FUNCTION_BLOCK TFCiclo_Deposito_Lastra
VAR_INPUT
	Ciclo 		: POINTER TO Stato_Ciclo_Lavoro;
	Programma 	: POINTER TO TFProgramma_Ciclo_Lastra;
	ModuleAX_X 	: POINTER TO TFModulePalletizer_Ax;
	ModuleAX_Y 	: POINTER TO TFModulePalletizer_Ax;
	ModuleAX_Z 	: POINTER TO TFModulePalletizer_Ax;
	ModuleAX_J 	: POINTER TO TFModulePalletizer_AxJ_Lastre;
	ModulePinza : POINTER TO TFModulePalletizer_Pinza;
	StartInterpolazioneAssi : POINTER TO BOOL;
	QuotaPassModePuntoIntermedio : ARRAY [1..3] OF REAL;
	AbilitazioneGlobalePassMode	: BOOL;
	InterrompiCiclo : BOOL;
	Abilita_Ciclo_Step : BOOL;
	Command_Step : BOOL;
	AbilitazioneAnticipoDinamicoMovimenti : BOOL;

END_VAR
VAR_OUTPUT
	STEPDone	: BOOL;
	Errore : UINT;
END_VAR
VAR
	ConAccostamentoZ : BOOL := FALSE;
	StepInto: BOOL;
	PinzaInPresa : BOOL;
	PinzaVerticale : BOOL;
END_VAR

(* Set della variabile che mi permette di fare lo STEP nel ciclo *)
TFTimerCall(ADR(ReMovEjeXCicloDeposito),TimeBase);
StepInto := (Abilita_Ciclo_Step AND Command_Step) OR NOT Abilita_Ciclo_Step;

(* Reset Anticipo Dinamico se non ho l'abilitazione *)
IF NOT AbilitazioneAnticipoDinamicoMovimenti OR NOT HMI_DisabilitaAnticipiGLOBALE THEN
	QuotaAnticipoDinamicaX_Raggiunta := FALSE;
	QuotaAnticipoDinamicaY_Raggiunta := FALSE;
	QuotaAnticipoDinamicaZ_Raggiunta := FALSE;
END_IF

PinzaInPresa 	:= ModulePinza^.StatoPinza.ElementoPrelevato AND  
					ModulePinza^.StatoPinza.LatoDxPiastrellaInPresa AND
					ModulePinza^.StatoPinza.LatoSxPiastrellaInPresa;

PinzaVerticale := NOT(ModuleAX_J^.Ax^.Status.ActPosition > 85 AND ModuleAX_J^.Ax^.Status.ActPosition < 95);

EjeYPosFueraIngombroCargado := TFAsseInFinestra(Posizione_Attuale :=  ModuleAX_Y^.Ax^.Status.ActPosition ,
 Posizione_Finale := Programma_Y[Y_PosFuoriIngombroVuotoLastra].Quota_Destinazione ,FinestraDiControllo := 30.0 );

EjeYPos0Ingombro :=  TFAsseInFinestra(Posizione_Attuale := ModuleAX_Y^.Ax^.Status.ActPosition ,
 Posizione_Finale := Programma_Y[Y_PosPasillo0grados].Quota_Destinazione ,FinestraDiControllo := 30.0 ) ;
 
EjeYPos180Ingombro := TFAsseInFinestra(Posizione_Attuale := ModuleAX_Y^.Ax^.Status.ActPosition ,
 Posizione_Finale := Programma_Y[Y_PosPasillo180grados].Quota_Destinazione ,FinestraDiControllo := 30.0 ) ;
 
 EjeyPosLentaCoger := TFAsseInFinestra(Posizione_Attuale := ModuleAX_Y^.Ax^.Status.ActPosition ,
 Posizione_Finale := Programma_Y[Y_PosStartLentaDepositoLastra].Quota_Destinazione ,FinestraDiControllo := 30.0 ) ;

IF Ciclo^.Passo = 27 THEN

TFTimerSet(ADR(ReMovEjeXCicloDeposito),1000, FALSE );	
ELSE
TFTimerSet(ADR(ReMovEjeX),1000, 
TFAsseInFinestra(Posizione_Attuale := ModuleAX_Y^.Ax^.Status.ActPosition ,
 Posizione_Finale := Programma_Y[Y_PosFuoriIngombroVuotoLastra].Quota_Destinazione ,FinestraDiControllo := 30.0 ) );	
END_IF
  Temp_Bool[69]:=TFAsseInFinestra (Posizione_Attuale := ModuleAX_Y^.Ax^.Status.ActPosition ,
 Posizione_Finale := Programma_Y[Y_PosFuoriIngombroVuotoLastra].Quota_Destinazione ,FinestraDiControllo := 30.0 );
IF NOT InterrompiCiclo THEN
	IF Ciclo^.Stato = TERMINATO OR Ciclo^.Stato = ANNULLATO THEN
		Ciclo^.Passo := 0;
	//ELSIF Ciclo^.Stato = INTERROTTO AND Ciclo^.Passo = 56 THEN
	//	Ciclo^.Passo := 56;
	ELSIF Ciclo^.Stato = INTERROTTO THEN//AND NOT Ciclo^.Passo = 56 THEN
		Ciclo^.Passo := 999;
	END_IF
	Ciclo^.Stato := IN_ESECUZIONE;
	CASE Ciclo^.Passo OF
			(* Case 0 *)
			0:  Ciclo^.Stato := IN_ESECUZIONE;
				Ciclo^.Passo := 10;
				Errore := 0;
				STEPDone := FALSE;
				
			(* Case 10 -  *)
			10:	MaterialeDepositatoSuLinea := FALSE;
				IF PinzaVerticale THEN
					Ciclo^.Passo := 25;
				ELSE
					Ciclo^.Passo := 20;
				END_IF
						
			(* Case 20 - PROGRAMMA[Z_PosFuoriIngombroCaricoLastra] ASSE Z -> TRASLAZIONE A QUOTA DI FUORI INGOMBRO CON lLASTRA A BORDO *)	
			20:	Ciclo^.Stato := IN_ESECUZIONE;
				IF StepInto THEN
					Programma_Z[Z_PosFuoriIngombroCaricoLastra].Stato 			:= DA_ESEGUIRE;
					Programma_Z[Z_PosFuoriIngombroCaricoLastra].InterpolaAsse 	:= NO_INTERPOLAZIONE_ASSE;
					ProgrammaToModule_Z 										:= Programma_Z[Z_PosFuoriIngombroCaricoLastra];
					Ciclo^.Passo := 21;
					STEPDone := FALSE;
				END_IF
				
			(* Case 21 - Attesa completamento del comando MOVETOPOS o del raggiungimento quota di Pre-Movimento se abilitata la funzione*)
			21: 
				IF Programma_Z[Z_PosFuoriIngombroCaricoLastra].Stato = INTERROTTO THEN
					Ciclo^.Passo := 21;		
				ELSIF Programma_Z[Z_PosFuoriIngombroCaricoLastra].Stato = TERMINATO OR
					Asse_Z_InFinestraDiPassMode THEN
					Ciclo^.Passo := 24; //
					STEPDone := TRUE;							
				END_IF
			
			(* Case 22 - Fuori ingombro J - NON usato in questa fase *)	
			22: IF Programma_Z[Z_PosFuoriIngombroCaricoLastra].Stato = INTERROTTO THEN
					 Ciclo^.Passo := 22;
				ELSIF Programma_Z[Z_PosFuoriIngombroCaricoLastra].Stato = TERMINATO OR 
						Asse_Z_InFinestraDiPassMode OR 
						QuotaAnticipoDinamicaZ_Raggiunta THEN
							IF StepInto AND Temp_Bool[3] THEN 
								Programma_J[J_PosFuoriIngombro].Stato 			:= DA_ESEGUIRE;
								Programma_J[J_PosFuoriIngombro].InterpolaAsse 	:= NO_INTERPOLAZIONE_ASSE;
								ProgrammaToModule_J		 						:= Programma_J[J_PosFuoriIngombro];
								Ciclo^.Passo := 23;
								STEPDone := FALSE;
							END_IF									
				END_IF
			
			(* Case 23 - Attesa completamento Fuori ingombro J *)	
			23: IF Programma_Z[Z_PosFuoriIngombroCaricoLastra].Stato = INTERROTTO OR 
					Programma_J[J_PosFuoriIngombro].Stato = INTERROTTO THEN
					 Ciclo^.Passo := 23;
				ELSIF (Programma_Z[Z_PosFuoriIngombroCaricoLastra].Stato = TERMINATO OR Asse_Z_InFinestraDiPassMode (*OR QuotaAnticipoDinamicaZ_Raggiunta*)) AND 
					(Programma_J[J_PosFuoriIngombro].Stato = TERMINATO OR Asse_J_InFinestraDiPassMode OR QuotaAnticipoDinamicaJ_Raggiunta) THEN
						Ciclo^.Passo := 24;
						STEPDone := TRUE;										
				END_IF	
							
				
			(* Case 24 - Scelgo in quale direzione devo muovermi per primo a seconda della disposizione delle postazioni *)	
			24:	
				IF Programma_Z[Z_PosFuoriIngombroCaricoLastra].Stato = INTERROTTO THEN
					Ciclo^.Passo := 21;	
				ELSE
					Ciclo^.Passo := 25;
				END_IF
					
		{Region "Dipsoizione postazioni lungo X"}		
			(* Case 25 - Vado a quota di fuori ingombro con Y e J *)
			25:	
						Temp_Bool[84] := ((WorkAreaState[PosRobot].Supporto.Tipologia = CAVALLETTO AND 
							workAreaState[Mission.PPlace].Supporto.Tipologia = BUNDLE)  OR MultiplesCavalletesReceta ) AND PosicionJOrigen <> PosicionJDestino  ;
					
				IF StepInto THEN
					IF PinzaVerticale THEN
						Programma_Z[Z_PosFuoriIngombroCaricoLastra].Stato 			:= DA_ESEGUIRE;
						Programma_Z[Z_PosFuoriIngombroCaricoLastra].InterpolaAsse 	:= INTERPOLAZIONE_ASSE;
						ProgrammaToModule_Z 										:= Programma_Z[Z_PosFuoriIngombroCaricoLastra];
					END_IF
					
					IF WorkAreaState[PosRobot].Supporto.Tipologia = BUNDLE  AND Programma_J[J_PosFuoriIngombro].Quota_Destinazione = 0 THEN
						(*
						//**********************************************************************
						Programma_Y[Y_PosPasillo0grados].Stato 				:= NON_ESEGUITO;
						Programma_Y[Y_PosPasillo180grados].Stato 			:= NON_ESEGUITO;
						Programma_Y[Y_PosFuoriIngombroCaricoLastra].Stato 	:= NON_ESEGUITO;
						//********************************************************************
						*)
  						Programma_Y[Y_PosgiroPieza].Stato 			:= DA_ESEGUIRE;
						Programma_Y[Y_PosgiroPieza].InterpolaAsse 	:= INTERPOLAZIONE_ASSE;
						ProgrammaToModule_Y 						:= Programma_Y[Y_PosgiroPieza];
						IF Temp_Bool[2] THEN 
							Ciclo^.Passo := 27;
							STEPDone := FALSE;
						END_IF
					ELSIF ((WorkAreaState[PosRobot].Supporto.Tipologia = CAVALLETTO AND 
							workAreaState[Mission.PPlace].Supporto.Tipologia = BUNDLE)  OR MultiplesCavalletesReceta ) AND  NuEstacionPiking <> 0  
								 THEN
							IF PosicionJActual = 0 THEN
								Programma_Y[Y_PosPasillo0grados].Stato 			:= DA_ESEGUIRE;
								Programma_Y[Y_PosPasillo0grados].InterpolaAsse 	:= INTERPOLAZIONE_ASSE;
								ProgrammaToModule_Y 							:= Programma_Y[Y_PosPasillo0grados];
								IF Temp_Bool[10] AND EjeYPos0Ingombro THEN 
									Ciclo^.Passo := 60;
									STEPDone := FALSE;
								END_IF
							END_IF
							IF PosicionJActual = 180  THEN
								Programma_Y[Y_PosPasillo180grados].Stato 			:= DA_ESEGUIRE;
								Programma_Y[Y_PosPasillo180grados].InterpolaAsse 	:= INTERPOLAZIONE_ASSE;
								ProgrammaToModule_Y 								:= Programma_Y[Y_PosPasillo180grados];
								IF Temp_Bool[10]AND EjeYPos180Ingombro THEN 
									Ciclo^.Passo := 60;
									STEPDone := FALSE;
								END_IF
							END_IF
							
							IF PosicionJActual = 90 THEN
								IF PosicionJDestino = 0 THEN
									Programma_Y[Y_PosPasillo0grados].Stato 			:= DA_ESEGUIRE;
									Programma_Y[Y_PosPasillo0grados].InterpolaAsse 	:= INTERPOLAZIONE_ASSE;
									ProgrammaToModule_Y 							:= Programma_Y[Y_PosPasillo0grados];
									
									Programma_J[Pos0TrasporteCavallete].Stato 						:= DA_ESEGUIRE;
									Programma_J[Pos0TrasporteCavallete].InterpolaAsse 				:= INTERPOLAZIONE_ASSE;
									ProgrammaToModule_J		 									:= Programma_J[Pos0TrasporteCavallete];
									
									IF Temp_Bool[10] AND EjeYPos0Ingombro THEN 
										Ciclo^.Passo := 60;
										STEPDone := FALSE;
									END_IF
								END_IF
								
								IF PosicionJDestino = 180  THEN
									Programma_Y[Y_PosPasillo180grados].Stato 			:= DA_ESEGUIRE;
									Programma_Y[Y_PosPasillo180grados].InterpolaAsse 	:= INTERPOLAZIONE_ASSE;
									ProgrammaToModule_Y 								:= Programma_Y[Y_PosPasillo180grados];
									
									Programma_J[Pos180TrasporteCavallete].Stato 						:= DA_ESEGUIRE;
									Programma_J[Pos180TrasporteCavallete].InterpolaAsse 				:= INTERPOLAZIONE_ASSE;
									ProgrammaToModule_J		 									:= Programma_J[Pos180TrasporteCavallete];
									
									IF Temp_Bool[10] AND EjeYPos180Ingombro THEN 
										Ciclo^.Passo := 60;
										STEPDone := FALSE;
									END_IF
								END_IF
								IF PosicionJDestino = 90  THEN//*************************************************
									Programma_Y[Y_PosFuoriIngombroCaricoLastra].Stato 			:= DA_ESEGUIRE;
									Programma_Y[Y_PosFuoriIngombroCaricoLastra].InterpolaAsse 	:= INTERPOLAZIONE_ASSE;
									ProgrammaToModule_Y 										:= Programma_Y[Y_PosFuoriIngombroCaricoLastra];
									
									
									Programma_J[J_PosFuoriIngombro].Stato 						:= DA_ESEGUIRE;
									Programma_J[J_PosFuoriIngombro].InterpolaAsse 				:= INTERPOLAZIONE_ASSE;
									ProgrammaToModule_J		 									:= Programma_J[J_PosFuoriIngombro];
									
									StartInterpolazioneAssi^ := TRUE; //Abilito l'interpolazione degli assi						
									IF Temp_Bool[90] THEN 
											Ciclo^.Passo := 26;
											STEPDone := FALSE;
									END_IF
								END_IF
							END_IF
						
					
						
							
					ELSIF (((WorkAreaState[PosRobot].Supporto.Tipologia = CAVALLETTO AND 
							workAreaState[Mission.PPlace].Supporto.Tipologia = BUNDLE ) OR MultiplesCavalletesReceta) AND PosicionJOrigen = PosicionJDestino ) OR 
								(WorkAreaState[PosRobot].Supporto.Tipologia = CASSA_STANDARD AND 	
								WorkAreaState[Mission.PPlace].Supporto.Tipologia = CASSA_STANDARD AND 
									PosicionJActual = PosicionJDestino ) 
								 												THEN
						(*
						//********************************************************************++
						Programma_Y[Y_PosPasillo0grados].Stato 				:= NON_ESEGUITO;
						Programma_Y[Y_PosPasillo180grados].Stato 			:= NON_ESEGUITO;
						Programma_Y[Y_PosgiroPieza].Stato 					:= NON_ESEGUITO;		 
						//********************************************************************++	
						*)	 
						Programma_Y[Y_PosFuoriIngombroCaricoLastra].Stato 			:= DA_ESEGUIRE;
						Programma_Y[Y_PosFuoriIngombroCaricoLastra].InterpolaAsse 	:= INTERPOLAZIONE_ASSE;
						ProgrammaToModule_Y 										:= Programma_Y[Y_PosFuoriIngombroCaricoLastra];
						
						
						Programma_J[J_PosFuoriIngombro].Stato 						:= DA_ESEGUIRE;
						Programma_J[J_PosFuoriIngombro].InterpolaAsse 				:= INTERPOLAZIONE_ASSE;
						ProgrammaToModule_J		 									:= Programma_J[J_PosFuoriIngombro];
						
						StartInterpolazioneAssi^ := TRUE; //Abilito l'interpolazione degli assi						
						IF Temp_Bool[90] THEN 
						Ciclo^.Passo := 26;
						STEPDone := FALSE;
						END_IF
					ELSIF workAreaState[PosRobot].Supporto.Tipologia = BUNDLE  AND  PosicionJOrigen = PosicionJDestino  
								 THEN
						(*
						//********************************************************************++
						Programma_Y[Y_PosPasillo0grados].Stato 				:= NON_ESEGUITO;
						Programma_Y[Y_PosPasillo180grados].Stato 			:= NON_ESEGUITO;
						Programma_Y[Y_PosgiroPieza].Stato 					:= NON_ESEGUITO;		 
						//********************************************************************++
						*)	
						Programma_Y[Y_PosFuoriIngombroCaricoLastra].Stato 			:= DA_ESEGUIRE;
						Programma_Y[Y_PosFuoriIngombroCaricoLastra].InterpolaAsse 	:= INTERPOLAZIONE_ASSE;
						ProgrammaToModule_Y 										:= Programma_Y[Y_PosFuoriIngombroCaricoLastra];
						
						
						Programma_J[J_PosFuoriIngombro].Stato 						:= DA_ESEGUIRE;
						Programma_J[J_PosFuoriIngombro].InterpolaAsse 				:= INTERPOLAZIONE_ASSE;
						ProgrammaToModule_J		 									:= Programma_J[J_PosFuoriIngombro];
						
						StartInterpolazioneAssi^ := TRUE; //Abilito l'interpolazione degli assi						
						IF Temp_Bool[90] THEN 
						Ciclo^.Passo := 26;
						STEPDone := FALSE;
						END_IF
					ELSE
						(*
						//********************************************************************++
						Programma_Y[Y_PosPasillo0grados].Stato 				:= NON_ESEGUITO;
						Programma_Y[Y_PosPasillo180grados].Stato 			:= NON_ESEGUITO;
						Programma_Y[Y_PosgiroPieza].Stato 					:= NON_ESEGUITO;		 
						//********************************************************************++
						*)	
						Programma_Y[Y_PosFuoriIngombroCaricoLastra].Stato 			:= DA_ESEGUIRE;
						Programma_Y[Y_PosFuoriIngombroCaricoLastra].InterpolaAsse 	:= INTERPOLAZIONE_ASSE;
						ProgrammaToModule_Y 										:= Programma_Y[Y_PosFuoriIngombroCaricoLastra];
						
						
						Programma_J[J_PosFuoriIngombro].Stato 						:= DA_ESEGUIRE;
						Programma_J[J_PosFuoriIngombro].InterpolaAsse 				:= INTERPOLAZIONE_ASSE;
						ProgrammaToModule_J		 									:= Programma_J[J_PosFuoriIngombro];
						
						StartInterpolazioneAssi^ := TRUE; //Abilito l'interpolazione degli assi						
						IF Temp_Bool[90] THEN 
						Ciclo^.Passo := 26;
						STEPDone := FALSE;
						END_IF
					END_IF 
					
				END_IF
					
					
				
			// VOY CON X A LA POSICION DE DEPOSITO
			60: 	IF 
 						(Programma_Y[Y_PosPasillo0grados].Stato 				= INTERROTTO AND PosicionJActual = 0) OR 
						(Programma_Y[Y_PosPasillo180grados].Stato 			= INTERROTTO AND PosicionJActual = 180 )OR 
						Programma_Z[Z_PosFuoriIngombroCaricoLastra].Stato 	= INTERROTTO OR 
						Programma_J[J_PosSfogliatura].Stato 				= INTERROTTO THEN
						Ciclo^.Passo := 60;
					ELSE	
						IF  ((Programma_Y[Y_PosPasillo0grados].Stato 				= TERMINATO AND PosicionJActual = 0) OR  
							(Programma_Y[Y_PosPasillo180grados].Stato 			= TERMINATO AND PosicionJActual = 180)) AND
							Programma_Z[Z_PosFuoriIngombroCaricoLastra].Stato 	= TERMINATO AND
							Programma_J[J_PosSfogliatura].Stato 				= TERMINATO THEN
								 	
							IF 	NOT MultiplesCavalletesReceta OR PosicionJDestino = 90 OR (WorkAreaState[Mission.PPlace].Supporto.Tipologia = BUNDLE AND MultiplesCavalletesReceta) THEN	
							Programma_X[X_PosStartLentaDepositoLastra].Stato 			:= DA_ESEGUIRE;
							Programma_X[X_PosStartLentaDepositoLastra].InterpolaAsse 	:= NO_INTERPOLAZIONE_ASSE;
							ProgrammaToModule_X 										:= Programma_X[X_PosStartLentaDepositoLastra];
							ELSE 
								Programma_X[X_PosGiroPiezaTraCavallete].Stato 			:= DA_ESEGUIRE;
								Programma_X[X_PosGiroPiezaTraCavallete].InterpolaAsse 	:= NO_INTERPOLAZIONE_ASSE;
								ProgrammaToModule_X 										:= Programma_X[X_PosGiroPiezaTraCavallete];
							END_IF
							IF Temp_Bool[11] THEN 
								Ciclo^.Passo := 61;
								STEPDone := FALSE;	
							END_IF
						END_IF 
					END_IF	
			 // VPY CON Y A LA POSICION DE GIRAR		
					
			61: 	IF (Programma_Y[Y_PosFuoriIngombroCaricoLastra].Stato 	= INTERROTTO AND ProgramaEjes.EjeY = 127)  OR 
						(Programma_Y[Y_PosPasillo0grados].Stato 				= INTERROTTO  AND  PosicionJActual = 0 AND ProgramaEjes.EjeY = 128 )OR
						(Programma_Y[Y_PosPasillo180grados].Stato 				= INTERROTTO  AND  PosicionJActual = 180 AND  ProgramaEjes.EjeY = 129)OR
						Programma_Z[Z_PosFuoriIngombroCaricoLastra].Stato 		= INTERROTTO OR 
						Programma_J[J_PosSfogliatura].Stato 					= INTERROTTO OR
						(Programma_X[X_PosStartLentaDepositoLastra].Stato 		= INTERROTTO AND ProgramaEjes.EjeX = 104) OR 
						(Programma_X[X_PosGiroPiezaTraCavallete].Stato 			= INTERROTTO AND  ProgramaEjes.EjeX = 127) 	THEN
						Ciclo^.Passo := 60;
					ELSE	
						IF ((Programma_Y[Y_PosFuoriIngombroCaricoLastra].Stato =  TERMINATO AND ProgramaEjes.EjeY = 127 )OR
							(Programma_Y[Y_PosPasillo0grados].Stato =  TERMINATO AND   PosicionJActual = 0 AND ProgramaEjes.EjeY = 128) OR
							(Programma_Y[Y_PosPasillo180grados].Stato =  TERMINATO AND  PosicionJActual = 180 AND ProgramaEjes.EjeY = 129 ))
							AND	Programma_Z[Z_PosFuoriIngombroCaricoLastra].Stato = TERMINATO 
								AND	Programma_J[J_PosSfogliatura].Stato = TERMINATO
									AND ((Programma_X[X_PosStartLentaDepositoLastra].Stato =TERMINATO AND ProgramaEjes.EjeX = 104) OR
									 (Programma_X[X_PosGiroPiezaTraCavallete].Stato =TERMINATO AND ProgramaEjes.EjeX = 127 )) AND PosicionJDestino <> 90 		THEN
									 
									 
								IF (Programma_X[X_PosGiroPiezaTraCavallete].Stato =TERMINATO AND ProgramaEjes.EjeX = 127) OR  
									(Programma_X[X_PosStartLentaDepositoLastra].Stato 		= TERMINATO AND ProgramaEjes.EjeX = 104 AND PosicionJActual <> PosicionJDestino)		THEN
									Programma_Y[Y_PosgiroPieza].Stato 			:= DA_ESEGUIRE;
									Programma_Y[Y_PosgiroPieza].InterpolaAsse 	:= INTERPOLAZIONE_ASSE;
									ProgrammaToModule_Y 						:= Programma_Y[Y_PosgiroPieza];
									IF Temp_Bool[12] THEN 
										Ciclo^.Passo := 62;
										STEPDone := FALSE;	
									END_IF
									ELSIF Programma_X[X_PosStartLentaDepositoLastra].Stato 		= TERMINATO AND ProgramaEjes.EjeX = 104 and PosicionJActual = PosicionJDestino THEN 
									IF Temp_Bool[12] THEN 
										Ciclo^.Passo := 31;
										STEPDone := FALSE;	
									END_IF	
								END_IF
							ELSIF  ((Programma_Y[Y_PosFuoriIngombroCaricoLastra].Stato =  TERMINATO AND ProgramaEjes.EjeY = 127 )OR
										(Programma_Y[Y_PosPasillo0grados].Stato =  TERMINATO AND   PosicionJActual = 0 AND ProgramaEjes.EjeY = 128) OR
											(Programma_Y[Y_PosPasillo180grados].Stato =  TERMINATO AND  PosicionJActual = 180 AND ProgramaEjes.EjeY = 129 ))
													AND	Programma_Z[Z_PosFuoriIngombroCaricoLastra].Stato = TERMINATO 
															AND	Programma_J[J_PosSfogliatura].Stato = TERMINATO
																AND ((Programma_X[X_PosStartLentaDepositoLastra].Stato =TERMINATO AND ProgramaEjes.EjeX = 104) OR
									 								(Programma_X[X_PosGiroPiezaTraCavallete].Stato =TERMINATO AND ProgramaEjes.EjeX = 127 )) AND PosicionJDestino = 90	 THEN 
										IF Temp_Bool[12] THEN 
										Ciclo^.Passo := 31;
										STEPDone := FALSE;	
									END_IF						
						END_IF 
					END_IF	
			62: 	IF Programma_Y[Y_PosgiroPieza].Stato 	= INTERROTTO  OR 
						Programma_Z[Z_PosFuoriIngombroCaricoLastra].Stato 	= INTERROTTO OR 
						Programma_J[J_PosSfogliatura].Stato 				= INTERROTTO OR
						Programma_X[X_PosStartLentaDepositoLastra].Stato 	= INTERROTTO AND NOT MultiplesCavalletesReceta OR 
						Programma_X[X_PosGiroPiezaTraCavallete].Stato 	= INTERROTTO AND MultiplesCavalletesReceta	 THEN
						Ciclo^.Passo := 62;
					ELSE	
						IF Programma_Y[Y_PosgiroPieza].Stato =  TERMINATO 	
								AND	Programma_Z[Z_PosFuoriIngombroCaricoLastra].Stato = TERMINATO 
									AND	Programma_J[J_PosSfogliatura].Stato = TERMINATO
									AND Programma_X[X_PosStartLentaDepositoLastra].Stato =TERMINATO AND NOT MultiplesCavalletesReceta OR 	
										Programma_X[X_PosGiroPiezaTraCavallete].Stato =TERMINATO AND  MultiplesCavalletesReceta	THEN
							Programma_J[J_PosFuoriIngombro].Stato 						:= DA_ESEGUIRE;
							Programma_J[J_PosFuoriIngombro].InterpolaAsse 				:= INTERPOLAZIONE_ASSE;
							ProgrammaToModule_J		 									:= Programma_J[J_PosFuoriIngombro];
							IF Temp_Bool[13] THEN 
								Ciclo^.Passo := 63;
								STEPDone := FALSE;	
							END_IF
						END_IF 
					END_IF	
			63: 	IF Programma_Y[Y_PosgiroPieza].Stato 	= INTERROTTO  OR 
						Programma_Z[Z_PosFuoriIngombroCaricoLastra].Stato 	= INTERROTTO OR 
						Programma_J[J_PosFuoriIngombro].Stato 				= INTERROTTO OR
						Programma_X[X_PosStartLentaDepositoLastra].Stato 	= INTERROTTO AND NOT MultiplesCavalletesReceta OR
						Programma_X[X_PosGiroPiezaTraCavallete].Stato =INTERROTTO AND  MultiplesCavalletesReceta THEN
						Ciclo^.Passo := 63;
					ELSE	
						IF Programma_Y[Y_PosgiroPieza].Stato =  TERMINATO 	
								AND	Programma_Z[Z_PosFuoriIngombroCaricoLastra].Stato = TERMINATO 
									AND	Programma_J[J_PosFuoriIngombro].Stato = TERMINATO
									AND (Programma_X[X_PosStartLentaDepositoLastra].Stato =TERMINATO AND NOT MultiplesCavalletesReceta) OR
									(Programma_X[X_PosGiroPiezaTraCavallete].Stato = TERMINATO AND  MultiplesCavalletesReceta )	THEN
						(*
						//********************************************************************++
						Programma_Y[Y_PosPasillo0grados].Stato 				:= NON_ESEGUITO;
						Programma_Y[Y_PosPasillo180grados].Stato 			:= NON_ESEGUITO;
						Programma_Y[Y_PosgiroPieza].Stato 					:= NON_ESEGUITO;		 
						//********************************************************************++
						*)	
							Programma_Y[Y_PosFuoriIngombroCaricoLastra].Stato 			:= DA_ESEGUIRE;
							Programma_Y[Y_PosFuoriIngombroCaricoLastra].InterpolaAsse 	:= INTERPOLAZIONE_ASSE;
							ProgrammaToModule_Y 										:= Programma_Y[Y_PosFuoriIngombroCaricoLastra];
							IF Temp_Bool[14] THEN 
								Ciclo^.Passo := 64;
								STEPDone := FALSE;	
							END_IF
						END_IF 
					END_IF	
			64 :
				 IF Programma_X[X_PosStartLentaDepositoLastra].Stato = INTERROTTO AND NOT MultiplesCavalletesReceta OR
					Programma_X[X_PosGiroPiezaTraCavallete].Stato = INTERROTTO AND  MultiplesCavalletesReceta OR 
					Programma_Y[Y_PosFuoriIngombroCaricoLastra].Stato = INTERROTTO OR
					Programma_Z[Z_PosFuoriIngombroCaricoLastra].Stato = INTERROTTO OR 
					Programma_J[J_PosFuoriIngombro].Stato = INTERROTTO THEN
						Ciclo^.Passo := 64;
				ELSE	
						IF (Programma_Y[Y_PosFuoriIngombroCaricoLastra].Stato =  TERMINATO AND ProgramaEjes.EjeY = 126) AND 	
							Programma_Z[Z_PosFuoriIngombroCaricoLastra].Stato = TERMINATO AND
							Programma_J[J_PosFuoriIngombro].Stato = TERMINATO AND 
									((Programma_X[X_PosStartLentaDepositoLastra].Stato =TERMINATO AND NOT MultiplesCavalletesReceta) OR
									(Programma_X[X_PosGiroPiezaTraCavallete].Stato = TERMINATO AND  MultiplesCavalletesReceta ) )AND  Temp_Bool[69] AND  Temp_Bool[70]	THEN
							Programma_X[X_PosStartLentaDepositoLastra].Stato 			:= DA_ESEGUIRE;
							Programma_X[X_PosStartLentaDepositoLastra].InterpolaAsse 	:= NO_INTERPOLAZIONE_ASSE;
							ProgrammaToModule_X 										:= Programma_X[X_PosStartLentaDepositoLastra];
							IF Temp_Bool[18] THEN 
								Ciclo^.Passo := 31;
								STEPDone := FALSE;	
							END_IF
						END_IF 
				END_IF	
			
					
			27: 	IF Programma_Y[Y_PosgiroPieza].Stato 	= INTERROTTO  OR 
						Programma_Z[Z_PosFuoriIngombroCaricoLastra].Stato 	= INTERROTTO OR 
						Programma_J[J_PosFuoriIngombro].Stato 				= INTERROTTO THEN
						Ciclo^.Passo := 27;
					ELSE	
						IF Programma_Y[Y_PosgiroPieza].Stato =  TERMINATO 		THEN
							Programma_J[J_PosFuoriIngombro].Stato 						:= DA_ESEGUIRE;
							Programma_J[J_PosFuoriIngombro].InterpolaAsse 				:= No_INTERPOLAZIONE_ASSE;
							ProgrammaToModule_J		 									:= Programma_J[J_PosFuoriIngombro];
							IF Temp_Bool[11] THEN 
							Ciclo^.Passo := 28;
							STEPDone := FALSE;	
					END_IF
						END_IF 
					END_IF
					
			28: 	IF Programma_Y[Y_PosgiroPieza].Stato 	= INTERROTTO  OR 
						Programma_Z[Z_PosFuoriIngombroCaricoLastra].Stato 	= INTERROTTO OR 
						Programma_J[J_PosFuoriIngombro].Stato 				= INTERROTTO THEN
						Ciclo^.Passo := 27;
					ELSE	
						IF Programma_Y[Y_PosgiroPieza].Stato =  TERMINATO AND Programma_J[J_PosFuoriIngombro].Stato = TERMINATO	 	THEN
							
						(*
						//********************************************************************++
						Programma_Y[Y_PosPasillo0grados].Stato 				:= NON_ESEGUITO;
						Programma_Y[Y_PosPasillo180grados].Stato 			:= NON_ESEGUITO;
						Programma_Y[Y_PosgiroPieza].Stato 					:= NON_ESEGUITO;		 
						//********************************************************************++
						*)	
							Programma_Y[Y_PosFuoriIngombroCaricoLastra].Stato 			:= DA_ESEGUIRE;
							Programma_Y[Y_PosFuoriIngombroCaricoLastra].InterpolaAsse 	:= INTERPOLAZIONE_ASSE;
							ProgrammaToModule_Y 										:= Programma_Y[Y_PosFuoriIngombroCaricoLastra];
							IF Temp_Bool[12] THEN 
							Ciclo^.Passo := 26;
							STEPDone := FALSE;	
							END_IF
						END_IF 
					END_IF
					
			(* Case 26 - Check se a quota di fuori ingombro con Y & J *)		
			26:	IF Programma_Y[Y_PosFuoriIngombroCaricoLastra].Stato 	= INTERROTTO OR 
					Programma_Z[Z_PosFuoriIngombroCaricoLastra].Stato 	= INTERROTTO OR 
					Programma_J[J_PosFuoriIngombro].Stato 				= INTERROTTO THEN
						Ciclo^.Passo := 26;
				ELSE	
				IF WorkAreaState[PosRobot].Supporto.Tipologia = BUNDLE  AND Programma_J[J_PosFuoriIngombro].Quota_Destinazione = 0 THEN
					IF  Programma_Y[Y_PosFuoriIngombroCaricoLastra].Stato = TERMINATO  AND
						Programma_J[J_PosFuoriIngombro].Stato = TERMINATO  AND
						Programma_Z[Z_PosFuoriIngombroCaricoLastra].Stato = TERMINATO THEN
						IF Temp_Bool[91] THEN 
						Ciclo^.Passo := 30;
						STEPDone := TRUE;	
						END_IF						
					END_IF
				ELSE
					IF (Programma_Y[Y_PosFuoriIngombroCaricoLastra].Stato = TERMINATO OR Asse_Y_InFinestraDiPassMode OR QuotaAnticipoDinamicaY_Raggiunta) AND
						(Programma_J[J_PosFuoriIngombro].Stato = TERMINATO OR Asse_J_InFinestraDiPassMode OR QuotaAnticipoDinamicaJ_Raggiunta) AND
						Programma_Z[Z_PosFuoriIngombroCaricoLastra].Stato = TERMINATO THEN
						IF Temp_Bool[92] THEN 
						Ciclo^.Passo := 30;
						STEPDone := TRUE;	
						END_IF
					END_IF
				END_IF	
				END_IF
										
			(* Case 30 - PROGRAMMA[0] ASSE X  -> TRASLAZIONE A QUOTA DI DEPOSITO  *)	
			30:	IF Programma_Z[Z_PosFuoriIngombroCaricoLastra].Stato = INTERROTTO OR 
					Programma_Y[Y_PosFuoriIngombroCaricoLastra].Stato = INTERROTTO OR 
					Programma_J[J_PosFuoriIngombro].Stato = INTERROTTO THEN
						Ciclo^.Passo := 30;										
				ELSE
					IF StepInto THEN
						Programma_X[X_PosStartLentaDepositoLastra].Stato 			:= DA_ESEGUIRE;
						Programma_X[X_PosStartLentaDepositoLastra].InterpolaAsse 	:= NO_INTERPOLAZIONE_ASSE;
						ProgrammaToModule_X 										:= Programma_X[X_PosStartLentaDepositoLastra];
						IF Temp_Bool[93] THEN 
						Ciclo^.Passo := 31;
						STEPDone := FALSE;
						END_IF
					END_IF
				END_IF			
			
			(* Case 31 -  Attesa completamento del comando MOVETOPOS o del raggiungimento quota di Pre-Movimento se abilitata la funzione *)
			31: 
				IF Programma_X[X_PosStartLentaDepositoLastra].Stato = INTERROTTO   OR
					(Programma_Y[Y_PosFuoriIngombroCaricoLastra].Stato = INTERROTTO AND  ProgramaEjes.EjeY = 126 ) OR
					(Programma_Y[Y_PosPasillo0grados].Stato = INTERROTTO AND  ProgramaEjes.EjeY = 128)  OR
					(Programma_Y[Y_PosPasillo180grados].Stato = INTERROTTO AND  ProgramaEjes.EjeY = 129)  OR
					Programma_Z[Z_PosFuoriIngombroCaricoLastra].Stato = INTERROTTO OR 
					Programma_J[J_PosFuoriIngombro].Stato = INTERROTTO THEN
						Ciclo^.Passo := 31;
				ELSE	
					IF (Programma_X[X_PosStartLentaDepositoLastra].Stato = TERMINATO OR Asse_X_InFinestraDiPassMode OR QuotaAnticipoDinamicaX_Raggiunta) THEN 
						IF WorkAreaState[Mission.PPlace].Supporto.Tipologia <> CAVALLETTO AND WorkAreaState[Mission.PPlace].Supporto.Tipologia <> BUNDLE THEN //se non devo depositare nel cavalletto...	
							Ciclo^.Passo := 32;//ciclo per orizzontale
						ELSE
							Ciclo^.Passo := 40;//Ciclo per cavalletto
						END_IF
						STEPDone := TRUE;							
					END_IF
				END_IF
				
			(* Case 32 - Vado a quota di START LENTA CON GLI ASSI con Y,Z,J *)
			32:
				IF Programma_X[X_PosStartLentaDepositoLastra].Stato = INTERROTTO OR
					(Programma_Y[Y_PosFuoriIngombroCaricoLastra].Stato = INTERROTTO AND  ProgramaEjes.EjeY = 126 ) OR
					(Programma_Y[Y_PosPasillo0grados].Stato = INTERROTTO AND  ProgramaEjes.EjeY = 128)  OR
					(Programma_Y[Y_PosPasillo180grados].Stato = INTERROTTO AND  ProgramaEjes.EjeY = 129)  OR
					Programma_Z[Z_PosFuoriIngombroCaricoLastra].Stato = INTERROTTO OR 
					Programma_J[J_PosFuoriIngombro].Stato = INTERROTTO THEN
						Ciclo^.Passo := 32;										
				ELSE
					IF StepInto AND Programma_X[X_PosStartLentaDepositoLastra].Stato = TERMINATO  THEN
						TFParametersArrayClear(ADR(ParametersArray));
						Programma_Y[Y_PosStartLentaDepositoLastra].Stato 			:= DA_ESEGUIRE;
						Programma_Y[Y_PosStartLentaDepositoLastra].InterpolaAsse 	:= INTERPOLAZIONE_ASSE;
						ProgrammaToModule_Y 										:= Programma_Y[Y_PosStartLentaDepositoLastra];
				
						//Programma_Z[Z_PosStartLentaDepositoLastra].Stato 			:= DA_ESEGUIRE;
						//Programma_Z[Z_PosStartLentaDepositoLastra].InterpolaAsse 	:= INTERPOLAZIONE_ASSE;
						//ProgrammaToModule_Z 										:= Programma_Z[Z_PosStartLentaDepositoLastra];
						
						Programma_J[J_PosDepositoLastra].Stato 						:= DA_ESEGUIRE;
						Programma_J[J_PosDepositoLastra].InterpolaAsse 				:= INTERPOLAZIONE_ASSE;
						ProgrammaToModule_J 										:= Programma_J[J_PosDepositoLastra];
						
						StartInterpolazioneAssi^ := TRUE; //Abilito l'interpolazione degli assi
												
						Ciclo^.Passo := 33;
						STEPDone := FALSE;
					END_IF
				END_IF
			
			(* Case 33 - Attendo completamento comando o assi in finsetra *)
			33:
				IF Programma_Y[Y_PosStartLentaDepositoLastra].Stato 	= TERMINATO OR ((Asse_Y_InFinestraDiPassMode OR TRUE) AND WorkAreaState[Mission.PPlace].Supporto.Tipologia <> CAVALLETTO AND WorkAreaState[Mission.PPlace].Supporto.Tipologia <> BUNDLE) AND 
					Programma_J[J_PosDepositoLastra].Stato 				= TERMINATO OR ((Asse_J_InFinestraDiPassMode OR TRUE) AND WorkAreaState[Mission.PPlace].Supporto.Tipologia <> CAVALLETTO AND WorkAreaState[Mission.PPlace].Supporto.Tipologia <> BUNDLE) AND
					Programma_X[X_PosStartLentaDepositoLastra].Stato 	= TERMINATO (*OR Asse_X_InFinestraDiPassMode)*)THEN// AND 
					//Programma_Z[Z_PosStartLentaDepositoLastra].Stato 	= TERMINATO (*OR Asse_Z_InFinestraDiPassMode)*) THEN
					IF EjeyPosLentaCoger THEN
						Programma_Z[Z_PosStartLentaDepositoLastra].Stato 			:= DA_ESEGUIRE;
						Programma_Z[Z_PosStartLentaDepositoLastra].InterpolaAsse 	:= NO_INTERPOLAZIONE_ASSE;
						ProgrammaToModule_Z 										:= Programma_Z[Z_PosStartLentaDepositoLastra];			

						Ciclo^.Passo := 34;
						STEPDone := TRUE;
					END_IF
						
				ELSIF Programma_Y[Y_PosStartLentaDepositoLastra].Stato 	= INTERROTTO OR 
					Programma_J[J_PosDepositoLastra].Stato 				= INTERROTTO OR 
					Programma_X[X_PosStartLentaDepositoLastra].Stato 	= INTERROTTO THEN//OR
				//	Programma_Z[Z_PosStartLentaDepositoLastra].Stato 	= TERMINATO THEN
						Ciclo^.Passo := 33;								
				END_IF

			(* Case 34 - Vado a quota di finale con Z *)
			34:
				IF Programma_X[X_PosStartLentaDepositoLastra].Stato = INTERROTTO OR
					Programma_Y[Y_PosStartLentaDepositoLastra].Stato = INTERROTTO OR
					Programma_J[J_PosDepositoLastra].Stato = INTERROTTO OR 
					Programma_Z[Z_PosStartLentaDepositoLastra].Stato 	= INTERROTTO THEN
						Ciclo^.Passo := 34;										
				ELSE
					IF Programma_Z[Z_PosStartLentaDepositoLastra].Stato 	= TERMINATO THEN
						IF StepInto THEN
							TFParametersArrayClear(ADR(ParametersArray));
							//Programma_Y[Y_PosDepositoInLentaLastra].Stato 			:= DA_ESEGUIRE;
							//Programma_Y[Y_PosDepositoInLentaLastra].InterpolaAsse 	:= INTERPOLAZIONE_ASSE;
							//ProgrammaToModule_Y 									:= Programma_Y[Y_PosDepositoInLentaLastra];
					
							Programma_Z[Z_PosDepositoInLentaLastra].Stato 			:= DA_ESEGUIRE;
							Programma_Z[Z_PosDepositoInLentaLastra].InterpolaAsse 	:= NO_INTERPOLAZIONE_ASSE;
							ProgrammaToModule_Z 									:= Programma_Z[Z_PosDepositoInLentaLastra];
													
							StartInterpolazioneAssi^ := TRUE; //Abilito l'interpolazione degli assi
													
							Ciclo^.Passo := 35;
							STEPDone := FALSE;
						END_IF
					END_IF
				END_IF

			(* Case 35 - Attendo completamento comando o assi in finsetra *)
			35:
				IF 	Programma_Z[Z_PosDepositoInLentaLastra].Stato = TERMINATO (*OR Asse_Z_InFinestraDiPassMode)*) THEN
					Ciclo^.Passo := 90;
					STEPDone := TRUE;
				ELSIF Programma_Z[Z_PosDepositoInLentaLastra].Stato = INTERROTTO THEN
					Ciclo^.Passo := 35;								
				END_IF
		{endregion}

		{Region "CICLO CAVALLETTO"}							
			(* Case 40 - Vado a quota di START LENTA CON GLI ASSI con Y,Z *)
			40:
				IF Programma_X[X_PosStartLentaDepositoLastra].Stato = INTERROTTO OR
					Programma_Y[Y_PosFuoriIngombroCaricoLastra].Stato = INTERROTTO OR
					Programma_Z[Z_PosFuoriIngombroCaricoLastra].Stato = INTERROTTO OR 
					Programma_J[J_PosFuoriIngombro].Stato = INTERROTTO THEN
						Ciclo^.Passo := 40;										
				ELSE
					IF StepInto THEN
						TFParametersArrayClear(ADR(ParametersArray));
						Programma_Y[Y_PosStartLentaDepositoLastra].Stato 			:= DA_ESEGUIRE;
						Programma_Y[Y_PosStartLentaDepositoLastra].InterpolaAsse 	:= INTERPOLAZIONE_ASSE;
						ProgrammaToModule_Y 										:= Programma_Y[Y_PosStartLentaDepositoLastra];
				
						Programma_Z[Z_PosStartLentaDepositoLastra].Stato 			:= DA_ESEGUIRE;
						Programma_Z[Z_PosStartLentaDepositoLastra].InterpolaAsse 	:= INTERPOLAZIONE_ASSE;
						ProgrammaToModule_Z 										:= Programma_Z[Z_PosStartLentaDepositoLastra];
						
						Programma_J[J_PosDepositoLastra].Quota_Destinazione    		:= Programma_J[J_PosDepositoLastra].Quota_Destinazione;
						Programma_J[J_PosDepositoLastra].Stato 						:= DA_ESEGUIRE;
						Programma_J[J_PosDepositoLastra].InterpolaAsse 				:= NO_INTERPOLAZIONE_ASSE;
						ProgrammaToModule_J 										:= Programma_J[J_PosDepositoLastra];
						
						StartInterpolazioneAssi^ := TRUE; //Abilito l'interpolazione degli assi
												
						Ciclo^.Passo := 41;
						STEPDone := FALSE;
					END_IF
				END_IF
			
			(* Case 41 - Vado a quota di finale con Z *)
			41:
				

				IF Programma_X[X_PosStartLentaDepositoLastra].Stato = INTERROTTO OR
					Programma_Y[Y_PosStartLentaDepositoLastra].Stato = INTERROTTO OR
					Programma_J[J_PosDepositoLastra].Stato = INTERROTTO OR 
					Programma_Z[Z_PosStartLentaDepositoLastra].Stato 	= INTERROTTO THEN
						Ciclo^.Passo := 41;										
				ELSE
					IF Programma_Y[Y_PosStartLentaDepositoLastra].Stato = TERMINATO  AND
						Programma_J[J_PosDepositoLastra].Stato = TERMINATO AND
						Programma_Z[Z_PosStartLentaDepositoLastra].Stato = TERMINATO AND NOT STEPDone THEN
							STEPDone := TRUE;
					ELSIF STEPDone THEN 	
							IF StepInto THEN
								TFParametersArrayClear(ADR(ParametersArray));
								Programma_Y[Y_PosDepositoInLentaLastra].Stato 			:= DA_ESEGUIRE;
								Programma_Y[Y_PosDepositoInLentaLastra].InterpolaAsse 	:= INTERPOLAZIONE_ASSE;
								ProgrammaToModule_Y 									:= Programma_Y[Y_PosDepositoInLentaLastra];
						
								Programma_Z[Z_PosDepositoInLentaLastra].Stato 			:= DA_ESEGUIRE;
								Programma_Z[Z_PosDepositoInLentaLastra].InterpolaAsse 	:= INTERPOLAZIONE_ASSE;
								ProgrammaToModule_Z 									:= Programma_Z[Z_PosDepositoInLentaLastra];
														
								StartInterpolazioneAssi^ := TRUE; //Abilito l'interpolazione degli assi
														
								Ciclo^.Passo := 42;
								STEPDone := FALSE;
							END_IF
					END_IF
				END_IF
			
			(* Case 42 - Attesa completamento posizionamento di tutti gli assi e stacco aspirazione *)
			42: 
				IF Programma_X[X_PosStartLentaDepositoLastra].Stato = INTERROTTO OR
					Programma_Y[Y_PosDepositoInLentaLastra].Stato = INTERROTTO OR
					Programma_Z[Z_PosDepositoInLentaLastra].Stato 	= INTERROTTO THEN
						Ciclo^.Passo := 42;										
				ELSE
					IF Programma_Y[Y_PosDepositoInLentaLastra].Stato = TERMINATO AND
						Programma_Z[Z_PosDepositoInLentaLastra].Stato = TERMINATO AND NOT STEPDone THEN
						 STEPDone:= TRUE;
					ELSIF STEPDone THEN	
						IF StepInto THEN
							TFParametersArrayClear(ADR(ParametersArray));
							TFCommandSend(CmdUNLOAD,ParametersArray,ModulePinza^.Cmd);
							Ciclo^.Passo := 43;
							STEPDone := FALSE;
						END_IF	
					END_IF						
				END_IF

			(* Case 43 - Attesa completamento rilascio pezzo *)	
			43:
				IF TFStateCodeGet(ModulePinza^.State) = StateError THEN
					Ciclo^.Passo := 43;																
				ELSE
					STEPDone := TRUE;
					IF TFStateCodeGet(ModulePinza^.State) = StateUNLOAD_END THEN//Pezzo rilasciato
						Ciclo^.Passo := 45;//
					END_IF	
				END_IF

			(* Case 44 - Vado a quota di finale con J *)
			44:
				IF Programma_X[X_PosStartLentaDepositoLastra].Stato = INTERROTTO OR
					Programma_Y[Y_PosDepositoInLentaLastra].Stato = INTERROTTO OR
					Programma_Z[Z_PosDepositoInLentaLastra].Stato 	= INTERROTTO THEN
						Ciclo^.Passo := 44;										
				ELSE
					IF Programma_Y[Y_PosDepositoInLentaLastra].Stato = TERMINATO AND
						Programma_Z[Z_PosDepositoInLentaLastra].Stato = TERMINATO THEN
							IF StepInto THEN
								TFParametersArrayClear(ADR(ParametersArray));
								Programma_J[J_PosDepositoLastra].Stato 						:= DA_ESEGUIRE;
								Programma_J[J_PosDepositoLastra].InterpolaAsse 				:= NO_INTERPOLAZIONE_ASSE;
								ProgrammaToModule_J 										:= Programma_J[J_PosDepositoLastra];
								Ciclo^.Passo := 45;
								STEPDone := FALSE;
							END_IF
					END_IF
				END_IF

			(* Case 45 - Attendo completamento comando o assi in finsetra *)
			45:
				//IF Programma_J[J_PosDepositoLastra].Stato = TERMINATO THEN
				IF StepInto THEN	
					//********************************************************************++
						Programma_Y[Y_PosPasillo0grados].Stato 				:= NON_ESEGUITO;
						Programma_Y[Y_PosPasillo180grados].Stato 			:= NON_ESEGUITO;
						Programma_Y[Y_PosgiroPieza].Stato 					:= NON_ESEGUITO;		 
						//********************************************************************++	
				
					Programma_Y[Y_PosFuoriIngombroCaricoLastra].Stato 			:= DA_ESEGUIRE;
					Programma_Y[Y_PosFuoriIngombroCaricoLastra].InterpolaAsse 	:= NO_INTERPOLAZIONE_ASSE;
					ProgrammaToModule_Y 										:= Programma_Y[Y_PosFuoriIngombroCaricoLastra];
			
					Programma_Z[Z_PosFuoriIngombroCaricoLastra].Stato 			:= DA_ESEGUIRE;
					Programma_Z[Z_PosFuoriIngombroCaricoLastra].InterpolaAsse 	:= NO_INTERPOLAZIONE_ASSE;
					ProgrammaToModule_Z 										:= Programma_Z[Z_PosFuoriIngombroCaricoLastra];
				
					//Programma_J[J_PosFuoriIngombro].Stato 						:= DA_ESEGUIRE;
					//Programma_J[J_PosFuoriIngombro].InterpolaAsse 				:= INTERPOLAZIONE_ASSE;
					//ProgrammaToModule_J		 									:= Programma_J[J_PosFuoriIngombro];
					Ciclo^.Passo := 46;	
					STEPDone := FALSE;
				END_IF
				//ELSIF Programma_J[J_PosDepositoLastra].Stato = INTERROTTO THEN
				//	Ciclo^.Passo := 45;								
				//END_IF	

			(* Case 46 - Attendo completamento comando o assi in finsetra *)
			46:
				IF Programma_Z[Z_PosFuoriIngombroCaricoLastra].Stato = TERMINATO AND 
					Programma_Y[Y_PosFuoriIngombroCaricoLastra].Stato = TERMINATO THEN//AND
					//Programma_J[J_PosFuoriIngombro].Stato = TERMINATO THEN
						Ciclo^.Passo := 1000;	
						STEPDone := TRUE;
				ELSIF Programma_Z[Z_PosFuoriIngombroCaricoLastra].Stato = INTERROTTO AND  
					  Programma_Y[Y_PosFuoriIngombroCaricoLastra].Stato = INTERROTTO THEN
					Ciclo^.Passo := 46;								
				END_IF	
		{endregion}


		{Region "Dipsoizione postazioni lungo Y"}							
			(* Case 50 - Vado a quota di deposito con X *)
			50:	IF Programma_Z[Z_PosFuoriIngombroCaricoLastra].Stato = INTERROTTO OR
					Programma_J[J_PosFuoriIngombro].Stato = INTERROTTO THEN
						Ciclo^.Passo := 50;										
				ELSE
					IF StepInto THEN
						Programma_X[X_PosStartLentaDepositoLastra].Stato 			:= DA_ESEGUIRE;
						Programma_X[X_PosStartLentaDepositoLastra].InterpolaAsse 	:= NO_INTERPOLAZIONE_ASSE;
						ProgrammaToModule_X 										:= Programma_X[X_PosStartLentaDepositoLastra];
						Ciclo^.Passo := 51;
						STEPDone := FALSE;
					END_IF
				END_IF
					
			(* Case 51 - Check se a quota di deposito X *)		
			51:	IF Programma_X[X_PosStartLentaDepositoLastra].Stato = INTERROTTO OR 
					Programma_Z[Z_PosFuoriIngombroCaricoLastra].Stato = INTERROTTO OR 
					Programma_J[J_PosFuoriIngombro].Stato = INTERROTTO THEN
						Ciclo^.Passo := 51;
				ELSE	
					IF Programma_X[X_PosStartLentaDepositoLastra].Stato = TERMINATO OR 
						Asse_X_InFinestraDiPassMode THEN
							Ciclo^.Passo := 52;
							STEPDone := TRUE;							
					END_IF
				END_IF
										
			(* Case 52 - lancio posizionamento Y,j e x se non serve fuori ingombro  *)	
			52:	IF Programma_Z[Z_PosFuoriIngombroCaricoLastra].Stato = INTERROTTO OR 
					(Programma_X[X_PosStartLentaDepositoLastra].Stato = INTERROTTO AND FuoriIngombroXNecessario) OR 
					Programma_J[J_PosFuoriIngombro].Stato = INTERROTTO THEN
						Ciclo^.Passo := 52;										
				ELSE
					IF StepInto THEN
						IF NOT FuoriIngombroXNecessario THEN
							Programma_X[X_PosStartLentaDepositoLastra].Stato 			:= DA_ESEGUIRE;
							Programma_X[X_PosStartLentaDepositoLastra].InterpolaAsse 	:= INTERPOLAZIONE_ASSE;
							ProgrammaToModule_X 										:= Programma_X[X_PosStartLentaDepositoLastra];
						END_IF
					
						Programma_Y[Y_PosStartLentaDepositoLastra].Stato 			:= DA_ESEGUIRE;
						Programma_Y[Y_PosStartLentaDepositoLastra].InterpolaAsse 	:= INTERPOLAZIONE_ASSE;
						ProgrammaToModule_Y 										:= Programma_Y[Y_PosStartLentaDepositoLastra];
						
						//Programma_Z[Z_PosStartLentaDepositoLastra].Stato 			:= DA_ESEGUIRE;
						//Programma_Z[Z_PosStartLentaDepositoLastra].InterpolaAsse 	:= INTERPOLAZIONE_ASSE;
						//ProgrammaToModule_Z 										:= Programma_Z[Z_PosStartLentaDepositoLastra];
					
					
						Programma_J[J_PosDepositoLastra].Stato 						:= DA_ESEGUIRE;
						Programma_J[J_PosDepositoLastra].InterpolaAsse 				:= INTERPOLAZIONE_ASSE;
						ProgrammaToModule_J 										:= Programma_J[J_PosDepositoLastra];
			
						StartInterpolazioneAssi^ := TRUE; //Abilito l'interpolazione degli assi

						Ciclo^.Passo := 53;
						STEPDone := FALSE;
					END_IF
				END_IF			
				
			(* Case 53 -  Attesa completamento del comando MOVETOPOS o del raggiungimento quota di Pre-Movimento se abilitata la funzione *)
			53: 
				IF Programma_X[X_PosStartLentaDepositoLastra].Stato = INTERROTTO OR
					Programma_Y[Y_PosStartLentaDepositoLastra].Stato = INTERROTTO OR
					Programma_Z[Z_PosFuoriIngombroCaricoLastra].Stato = INTERROTTO OR 
					Programma_J[J_PosDepositoLastra].Stato = INTERROTTO THEN
						Ciclo^.Passo := 53;
				ELSE	
					IF (Programma_Y[Y_PosStartLentaDepositoLastra].Stato = TERMINATO OR Asse_Y_InFinestraDiPassMode OR QuotaAnticipoDinamicaY_Raggiunta) AND
						(Programma_J[J_PosDepositoLastra].Stato = TERMINATO OR Asse_J_InFinestraDiPassMode OR QuotaAnticipoDinamicaJ_Raggiunta)  THEN 
							
							Ciclo^.Passo := 54;
							STEPDone := TRUE;							
					END_IF
				END_IF
				
			(* Case 54 - Vado a quota di START LENTA CON GLI ASSI Z*)
			54:
				IF Programma_X[X_PosStartLentaDepositoLastra].Stato = INTERROTTO OR
					Programma_Y[Y_PosStartLentaDepositoLastra].Stato = INTERROTTO OR
					//Programma_Z[Z_PosStartLentaDepositoLastra].Stato = INTERROTTO OR 
					Programma_J[J_PosDepositoLastra].Stato = INTERROTTO THEN
						Ciclo^.Passo := 54;										
				ELSE
					IF StepInto THEN
						Programma_Z[Z_PosStartLentaDepositoLastra].Stato 			:= DA_ESEGUIRE;
						Programma_Z[Z_PosStartLentaDepositoLastra].InterpolaAsse 	:= NO_INTERPOLAZIONE_ASSE;
						ProgrammaToModule_Z 										:= Programma_Z[Z_PosStartLentaDepositoLastra];
								
						Ciclo^.Passo := 55;
						STEPDone := FALSE;
					END_IF
				END_IF
			
			(* Case 55 - Attendo completamento comando o assi in finsetra *)
			55:
				IF Programma_Y[Y_PosStartLentaDepositoLastra].Stato = TERMINATO (*OR Asse_Y_InFinestraDiPassMode)*) AND 
					Programma_J[J_PosDepositoLastra].Stato = TERMINATO (*OR Asse_J_InFinestraDiPassMode)*) AND
					Programma_X[X_PosStartLentaDepositoLastra].Stato = TERMINATO (*OR Asse_X_InFinestraDiPassMode)*) AND 
					Programma_Z[Z_PosStartLentaDepositoLastra].Stato = TERMINATO OR Asse_Z_InFinestraDiPassMode THEN
						Ciclo^.Passo := 56;
						STEPDone := TRUE;
				ELSIF Programma_X[X_PosStartLentaDepositoLastra].Stato = INTERROTTO OR
					Programma_Y[Y_PosStartLentaDepositoLastra].Stato = INTERROTTO OR
					Programma_Z[Z_PosFuoriIngombroCaricoLastra].Stato = INTERROTTO OR 
					Programma_J[J_PosDepositoLastra].Stato = INTERROTTO THEN
						Ciclo^.Passo := 55;
				END_IF

			(* Case 56 - Vado a quota di finale con Y,Z,J *)
			56:
				IF Programma_X[X_PosStartLentaDepositoLastra].Stato = INTERROTTO OR
					Programma_Y[Y_PosFuoriIngombroCaricoLastra].Stato = INTERROTTO OR
					Programma_Z[Z_PosFuoriIngombroCaricoLastra].Stato = INTERROTTO OR 
					Programma_J[J_PosFuoriIngombro].Stato = INTERROTTO THEN
						Ciclo^.Passo := 56;										
				ELSE
					IF StepInto THEN
						TFParametersArrayClear(ADR(ParametersArray));
						Programma_Z[Z_PosDepositoInLentaLastra].Stato 			:= DA_ESEGUIRE;
						Programma_Z[Z_PosDepositoInLentaLastra].InterpolaAsse 	:= NO_INTERPOLAZIONE_ASSE;
						ProgrammaToModule_Z 									:= Programma_Z[Z_PosDepositoInLentaLastra];						
						Ciclo^.Passo := 57;
						STEPDone := FALSE;						
						//StartInterpolazioneAssi^ := TRUE; //Abilito l'interpolazione degli assi
						
					END_IF
				END_IF

			(* Case 57 - Attendo completamento comando o assi in finsetra *)
			57:
				IF //Programma_Y[Y_PosStartLentaDepositoLastra].Stato = TERMINATO (*OR Asse_Y_InFinestraDiPassMode)*) AND 
					//Programma_J[J_PosDepositoLastra].Stato = TERMINATO (*OR Asse_J_InFinestraDiPassMode)*) AND
					//Programma_X[X_PosStartLentaDepositoLastra].Stato = TERMINATO (*OR Asse_X_InFinestraDiPassMode)*) AND 
					Programma_Z[Z_PosDepositoInLentaLastra].Stato = TERMINATO (*OR Asse_Z_InFinestraDiPassMode)*) THEN
						Ciclo^.Passo := 90;
						STEPDone := TRUE;
				ELSIF //Programma_Y[Y_PosStartLentaDepositoLastra].Stato = INTERROTTO OR 
					//Programma_J[J_PosDepositoLastra].Stato = INTERROTTO OR 
					//Programma_X[X_PosStartLentaDepositoLastra].Stato = INTERROTTO OR
					Programma_Z[Z_PosDepositoInLentaLastra].Stato = INTERROTTO THEN
					Ciclo^.Passo := 57;								
				END_IF
						
		{endregion}	
			(* Case 90 - Attesa completamento posizionamento di tutti gli assi *)
			90: 
				IF TFStateCodeGet(ModulePinza^.State) = StateError THEN
					Ciclo^.Passo := 90;																
				ELSE
					IF StepInto THEN
						TFParametersArrayClear(ADR(ParametersArray));
						TFCommandSend(CmdUNLOAD,ParametersArray,ModulePinza^.Cmd);
						Ciclo^.Passo := 91;
						STEPDone := FALSE;
					END_IF							
				END_IF

			(* Case 91 - Attesa completamento rilascio pezzo *)	
			91:
				IF TFStateCodeGet(ModulePinza^.State) = StateError THEN
					Ciclo^.Passo := 91;																
				ELSE
					STEPDone := TRUE;
					IF TFStateCodeGet(ModulePinza^.State) = StateUNLOAD_END THEN//Pezzo rilasciato
						RichiestaDepositoALinea := FALSE;
						Ciclo^.Passo := 1000;//dichiaro il ciclo terminato
					END_IF	
				END_IF
			
			(* Case 1000 *)
			1000:
				RichiestaDepositoALinea := FALSE;
				StopDepositoPerArresto := FALSE;
				Ciclo^.Stato := TERMINATO;
				Ciclo^.Passo := 1000;
				
			(* Case 9999 - Ciclo NON annullato o NON terminato*)
			9999:
				Ciclo^.Stato := INTERROTTO;
				Ciclo^.Passo := 9999;
	ELSE						
		;
			
	END_CASE;
	(* controllo pinza in presa durante il ciclo *)  
	IF WorkAreaState[Mission.PPlace].Supporto.Tipologia <> CAVALLETTO AND WorkAreaState[Mission.PPlace].Supporto.Tipologia <> BUNDLE THEN
		IF Ciclo^.Passo >= 20 AND Ciclo^.Passo <= 90 THEN
			IF PinzaInPresa THEN
				 ;
			ELSE
				Errore := ErrLOADLOST;//Segnalo mancanza presenza pezzo
			END_IF
		END_IF
	ELSE
		IF Ciclo^.Passo >= 20 AND Ciclo^.Passo <= 42 THEN
			IF PinzaInPresa THEN
				 ;
			ELSE
				Errore := ErrLOADLOST;//Segnalo mancanza presenza pezzo
			END_IF
		END_IF
	END_IF
ELSE								//Se il ciclo deve essere interrotto, setto il suo nuovo stato
	Ciclo^.Stato := INTERROTTO;
END_IF

END_FUNCTION_BLOCK

(* stored: Version 1.1.0.1, ProductVersion 3.1.4024.11
   POU TFCiclo_Deposito_Lastra: Id {79574767-b5f8-456d-a833-ececfee2abe1}, SpecialFunc None *)
